{attribute 'GeneratedUsingTerminal: EK1122-0000-0018'}
{attribute addProperty BoxType "EK1122-0000-0018"}
{attribute addProperty Id "Beckhoff_EL4xxxsub_EK1100EK1100_1FC0878B2"}
{attribute addProperty CRC "608164262"}
{attribute addProperty Size "2"}
TYPE Beckhoff_EL4xxxEK1122_243FD9A6 EXTENDS EK1122_1FC0878B :
STRUCT
	{attribute addProperty Name "Beckhoff_EL4xxxsub_EK1100"}
	{attribute addProperty PreviousPort "Beckhoff EL4xxxEK1122 : D"}
	Beckhoff_EL4xxxsub_EK1100 : EK1100_1FC0878B;
END_STRUCT
END_TYPE

(* stored: Version 1.2.0.0, ProductVersion 3.1.4024.9
   DUT Beckhoff_EL4xxxEK1122_243FD9A6: Id {dcb695ab-8c97-482d-92fa-eb2edb8a28d6} *)
